{attribute 'qualified_only'}
VAR_GLOBAL
END_VAR

(* stored: Version 1.1.0.1, ProductVersion 3.1.4022.7
   GVL GVL_02_Parameter_Servo_Motor_Shelf_Z: Id {4c0cf452-7ba1-436c-b7e0-eb1e9c8d4dd7} *)
